Staubli VAL3: decodeVelCmd.pgx

public program decodeVelCmd(bool& x_bFlag (dimensions=1))
  local num l_nIndex
  local num l_nRetVal
begin
  // Copyright (c) 2021, Institute for Factory Automation and Production Systems (FAPS)
  //
  // Licensed under the Apache License, Version 2.0 (the "License");
  // you may not use this file except in compliance with the License.
  // You may obtain a copy of the License at
  //
  //     http://www.apache.org/licenses/LICENSE-2.0
  //
  // Unless required by applicable law or agreed to in writing, software
  // distributed under the License is distributed on an "AS IS" BASIS,
  // WITHOUT WARRANTIES OR CONDITIONS OF ANY KIND, either express or implied.
  // See the License for the specific language governing permissions and
  // limitations under the License.


  // decode velocity command message body (data)

  // assume failure to decode
  velCmdAck.header.nReplyCode=SimpleMsg:ReplyCode.FAILURE


  // sequence, 4 bytes
  l_nRetVal=fromBinary(velCmdMsg.body.nData,4,"-4l",velCmdMsg.velCmd.nSeq)
  if (l_nRetVal!=1)
    x_bFlag=false
    return
  endIf

  // velocity vector [6], 24 bytes
  for l_nIndex=0 to 5 step 1
    l_nRetVal=fromBinary(velCmdMsg.body.nData[(l_nIndex*4)+4],4,"4.0l",velCmdMsg.velCmd.nVelVec[l_nIndex])
    if (l_nRetVal!=1)
      x_bFlag=false
      return
    endIf
  endFor

  // velocity command type (see Staubli:VelocityType "enum"), 4 bytes
  l_nRetVal=fromBinary(velCmdMsg.body.nData[28],4,"4l",velCmdMsg.velCmd.nCmdType)
  if (l_nRetVal!=1)
    x_bFlag=false
    return
  endIf


  // decoding successful
  velCmdAck.header.nReplyCode=SimpleMsg:ReplyCode.SUCCESS
  velCmdAck.velCmd.nSeq=velCmdMsg.velCmd.nSeq
  x_bFlag=true
end
